# EPICS substitutions: mc13/tpmacApp/Db/autohome.substitutions
file "$(EPICS_BASE)/db/autohome.db"
{

pattern
{SYS,              DEV,                 PLC,  PORT  }
{"XF:23ID1-ES",  "{Dif:Lens-Ax:TopX}",      8,     P0    }
{"XF:23ID1-ES",  "{Dif:Lens-Ax:TopY}",      9,     P0    }
{"XF:23ID1-ES",  "{Dif:Lens-Ax:TopZ}",      10,    P0    }
{"XF:23ID1-ES",  "{Dif:Lens-Ax:BotX}",      11,    P0    }
{"XF:23ID1-ES",  "{Dif:Lens-Ax:BotY}",      12,    P0    }
{"XF:23ID1-ES",  "{Dif:Lens-Ax:BotZ}",      13,    P0    }
}
